	// Step 2: Debounce filter (for rising edge)
	// TON: Q=TRUE only if rawInverted stays TRUE for DebounceTime continuously
	// rawInverted=FALSE immediately sets Q=FALSE (falling edge is unfiltered)
	// Note: To also filter the falling edge, add TOF -- not implemented currently
	#tonDebounce(IN := #rawInverted,
	             PT := #DebounceTime);

	IF #DebounceTime > T#0ms THEN
	    #State := #tonDebounce.Q;   // Filtered signal
	ELSE
	    #State := #rawInverted;     // Unfiltered (when DebounceTime=0)
	END_IF;

	// Step 3: Edge detection (compare with previous scan)
	#RisingEdge := #State AND NOT #prevState;
	#FallingEdge := NOT #State AND #prevState;
	#prevState := #State;

END_FUNCTION_BLOCK

FUNCTION_BLOCK "FB_SpindleControl"
{ S7_Optimized_Access := 'TRUE' }
VERSION : 3.0
// =============================================================================
// 07_SpindleControl.scl
// FB_SpindleControl -- Spindle speed control (simplified)
//
// Purpose:
//   Controls the spindle in velocity mode using MC_MoveVelocity (PTO output).
//   VFD run direction: CW only -- no direction pin.
//   RunForward signal enables VFD run.
//
// â”€â”€â”€â”€â”€â”€â”€â”€â”€â”€â”€â”€â”€â”€â”€â”€â”€â”€â”€â”€â”€â”€â”€â”€â”€â”€â”€â”€â”€â”€â”€â”€â”€â”€â”€â”€â”€â”€â”€â”€â”€â”€â”€â”€â”€â”€â”€â”€â”€â”€â”€â”€â”€â”€â”€â”€â”€â”€â”€â”€â”€â”€â”€â”€â”€â”€â”€â”€â”€â”€â”€â”€â”€â”€â”€â”€â”€
// OPERATING RULES (enforced by the CALLER, not by this FB):
//
//   1. Set SetSpeed while RunCmd = FALSE.
//   2. Set RunCmd = TRUE  â†’ MC_MoveVelocity starts + RunForward goes TRUE.
//      Keep RunCmd TRUE for the entire run.
//   3. To stop:  set RunCmd = FALSE  â†’ RunForward goes FALSE, PTO halts.
//      Do NOT touch SetSpeed during stop.
//   4. To change speed:
//        a. RunCmd = FALSE  (spindle coasts / stops on VFD ramp)
//        b. Write new SetSpeed
//        c. RunCmd = TRUE   (spindle restarts at new speed)
//
// This FB does NOT add any delays or intermediate states.
// Timing handshakes (coast-down waits, PTO stabilise, etc.) are the CALLER's
// responsibility if they are needed.
//
// â”€â”€â”€â”€â”€â”€â”€â”€â”€â”€â”€â”€â”€â”€â”€â”€â”€â”€â”€â”€â”€â”€â”€â”€â”€â”€â”€â”€â”€â”€â”€â”€â”€â”€â”€â”€â”€â”€â”€â”€â”€â”€â”€â”€â”€â”€â”€â”€â”€â”€â”€â”€â”€â”€â”€â”€â”€â”€â”€â”€â”€â”€â”€â”€â”€â”€â”€â”€â”€â”€â”€â”€â”€â”€â”€â”€â”€
// Speed calculation:
//   effectiveSpeed = CLAMP(SetSpeed, MinSpeed, MaxSpeed)
//   PTO conversion: velocity (pulse/s) = effectiveRPM Ã— 500 / 60
//   MinSpeed and MaxSpeed are read from DB_Spindle.
//
// Error codes:
//   16#0502 -- MC_MoveVelocity runtime error
//
// States (Diag_SpindleState):
//   0   = IDLE     -- RunCmd FALSE, all outputs safe
//   20  = RUNNING  -- RunCmd TRUE, PTO active, RunForward TRUE
//   999 = ERROR    -- cleared by AckError or Reset
//
// Change log:
//   2026-05-09  Complete rewrite: RunCmd level input replaces Start/Stop edges.
//               Removed STARTING and STOPPING delay states and mid-run
//               velocity-change handshake.  Caller owns all sequencing.
//   2026-05-09  Previous version: 4-state machine (was 7-state before that).
// =============================================================================
   VAR_INPUT
      Enable : Bool;   // Drive power enable -- from bDrivesEnable; stays TRUE during normal operation
      RunCmd : Bool;   // Level signal: TRUE = run, FALSE = stop/idle.   Set speed first, then raise RunCmd.   Lower RunCmd to stop; do not change speed while RunCmd is TRUE.
      SetSpeed : Real;   // Commanded speed in RPM (set while RunCmd = FALSE)
      SpeedOverride : Real;   // Speed override % (100 = normal speed)
      Reset : Bool;   // Full system reset -- clears ERROR, returns to IDLE
      AckError : Bool;   // Acknowledge spindle error only (no full system reset needed)
   END_VAR

   VAR_OUTPUT
      Running : Bool;   // TRUE while RunCmd is TRUE and no error
      AtSpeed : Bool;   // TRUE when actual speed is within SpeedTolerance of commanded
      ActualSpeed : Real;   // Measured speed (RPM)
      CommandedSpeed : Real;   // Override-applied target speed (RPM)
      Error : Bool;   // Error active
      ErrorID : Word;   // Error code
      RunForward : Bool;   // VFD Run Forward digital output -- mirrors RunCmd (except in ERROR)
   END_VAR

   VAR_IN_OUT
      Axis_Spindle {InstructionName := 'TO_PositioningAxis'; LibVersion := '8.0'} : TO_PositioningAxis;   // Spindle Technology Object
   END_VAR

   VAR
      state : Int;   // 0 = IDLE, 20 = RUNNING, 999 = ERROR Speed calculation
      effectiveRPM : Real;   // RPM after override and clamping
      targetVelocity : Real;   // Velocity in pulse/s sent to MC_MoveVelocity Motion FB instances
      MC_Power_Inst {InstructionName := 'MC_Power'; LibVersion := '8.0'} : MC_Power;
      MC_MoveVelocity_Inst {InstructionName := 'MC_MoveVelocity'; LibVersion := '8.0'} : MC_MoveVelocity;   // Internal execute flag
      bMoveVelExec : Bool;   // AtSpeed helpers
      speedDiff : Real;
      speedPercent : Real;   // AckError edge detection
      prevAck : Bool;
      ackEdge : Bool;
   END_VAR


BEGIN

	// =========================================================================
	// 1. EDGE DETECTION
	// =========================================================================
	#ackEdge := #AckError AND NOT #prevAck;
	#prevAck := #AckError;

	// =========================================================================
	// 2. RESET (full system reset -- takes priority over everything)
	// =========================================================================
	IF #Reset THEN
	    #state := 0;
	    #Error := FALSE;
	    #ErrorID := 0;
	    #bMoveVelExec := FALSE;
	    #RunForward := FALSE;
	END_IF;

	// =========================================================================
	// 3. SPEED CALCULATION (runs every scan)
	// =========================================================================
	#effectiveRPM := #SetSpeed * (#SpeedOverride / 100.0);
	IF #effectiveRPM < "DB_Spindle".MinSpeed THEN
	    #effectiveRPM := "DB_Spindle".MinSpeed;
	END_IF;
	IF #effectiveRPM > "DB_Spindle".MaxSpeed THEN
	    #effectiveRPM := "DB_Spindle".MaxSpeed;
	END_IF;
	#CommandedSpeed := #effectiveRPM;
	#targetVelocity := #effectiveRPM * 500.0 / 60.0;  // RPM â†’ pulse/s

	// =========================================================================
	// 4. STATE MACHINE
	// =========================================================================
	CASE #state OF

	        // -----------------------------------------------------------------
	        // STATE 0: IDLE
	        // All outputs safe.  Transition to RUNNING when RunCmd goes TRUE.
	        // -----------------------------------------------------------------
	    0:
	        #Running := FALSE;
	        #AtSpeed := FALSE;
	        #bMoveVelExec := FALSE;
	        #RunForward := FALSE;

	        IF #RunCmd THEN
	            #bMoveVelExec := TRUE;  // pre-load velocity; RunForward still FALSE
	            #state := 10;
	        END_IF;

	        // -----------------------------------------------------------------
	        // STATE 10: PRELOAD
	        // Execute TRUE so the PTO frequency is stable before the VFD is
	        // enabled.  RunForward stays FALSE this scan; transitions to RUNNING
	        // on the very next scan.
	        // -----------------------------------------------------------------
	    10:
	        #Running := FALSE;
	        #AtSpeed := FALSE;
	        #bMoveVelExec := TRUE;
	        #RunForward := FALSE;
	        #state := 20;

	        // -----------------------------------------------------------------
	        // STATE 20: RUNNING
	        // RunCmd TRUE â†’ MC_MoveVelocity active, RunForward TRUE.
	        // The CALLER is responsible for sequencing (speed-change stops,
	        // coast-down waits, PTO-stabilise delays, etc.).
	        // Transition back to IDLE when RunCmd goes FALSE.
	        // -----------------------------------------------------------------
	    20:
	        IF NOT #RunCmd THEN
	            // Caller dropped RunCmd â†’ stop immediately
	            #Running := FALSE;
	            #AtSpeed := FALSE;
	            #bMoveVelExec := FALSE;
	            #RunForward := FALSE;
	            #state := 0;

	        ELSE
	            // Normal running
	            #Running := TRUE;
	            #bMoveVelExec := TRUE;
	            #RunForward := TRUE;

	            // AtSpeed check
	            #speedDiff := ABS(#ActualSpeed - #effectiveRPM);
	            #speedPercent := 0.0;
	            IF #effectiveRPM > 1.0 THEN
	                #speedPercent := (#speedDiff / #effectiveRPM) * 100.0;
	            END_IF;
	            #AtSpeed := (#speedPercent <= "DB_Spindle".SpeedTolerance);

	            // MC_MoveVelocity error check
	            IF #MC_MoveVelocity_Inst.Error THEN
	                #ErrorID := 16#0502;
	                #bMoveVelExec := FALSE;
	                #RunForward := FALSE;
	                "DB_Diagnostic".Spindle_TO_ErrorID := #MC_MoveVelocity_Inst.ErrorID;
	                "DB_Diagnostic".TO_ErrorText := "FC_TO_ErrorText"(Code := #MC_MoveVelocity_Inst.ErrorID);
	                "DB_Diagnostic".Error_Text := CONCAT(IN1 := 'Spindle move failed: ',
	                                                     IN2 := "DB_Diagnostic".TO_ErrorText);
	                "DB_Diagnostic".Error_Code := #ErrorID;
	                // Single-writer: report via queue -> FB_AlarmManager latches DB_Error and
	                // drives DB_HMI.ErrorText through the mirror. (The old direct ErrorText
	                // write here was overwritten by the mirror one scan later and the error
	                // never reached DB_Error/history at all.)
	                "FC_ReportError"(Code := #ErrorID,
	                                 Details := "DB_Diagnostic".Error_Text,
	                                 Source := 'Spindle');
	                "DB_HMI".ErrorDetail := CONCAT(IN1 := 'TO:', IN2 := "DB_Diagnostic".TO_ErrorText);
	                "DB_HMI".ErrorDetail_ES := CONCAT(IN1 := 'TO:', IN2 := "DB_Diagnostic".TO_ErrorText);
	                #state := 999;
	            END_IF;
	        END_IF;

	        // -----------------------------------------------------------------
	        // STATE 999: ERROR
	        // AckError: clears spindle error, returns to IDLE.
	        // Reset:    handled above (takes priority, clears everything).
	        // -----------------------------------------------------------------
	    999:
	        #Error := TRUE;
	        #Running := FALSE;
	        #AtSpeed := FALSE;
	        #bMoveVelExec := FALSE;
	        #RunForward := FALSE;

	        IF #ackEdge THEN
	            #Error := FALSE;
	            #ErrorID := 0;
	            #state := 0;
	            // DB_HMI error text is owned by FB_AlarmManager (mirror) â€” Ack clears it
	            // there; STATE_STOPPED clears ErrorDetail. No HMI writes from this FB.
	        END_IF;

	END_CASE;

	// =========================================================================
	// 5. MC_ FUNCTION BLOCK CALLS (every scan)
	// =========================================================================
	#MC_Power_Inst(
	               Axis := #Axis_Spindle,
	               Enable := #Enable
	);
	#MC_MoveVelocity_Inst(
	                      Axis := #Axis_Spindle,
	                      Execute := #bMoveVelExec,
	                      Velocity := #targetVelocity,
	                      Direction := 1              // CW only -- no direction pin
	);

	// Actual speed: TO velocity (pulse/s) â†’ RPM
	#ActualSpeed := ABS(#Axis_Spindle.ActualVelocity) * 60.0 / 500.0;

	// =========================================================================
	// 6. WRITE STATUS TO DB_Spindle (read by HMI and other FBs)
	// =========================================================================
	"DB_Spindle".IsRunning := #Running;
	"DB_Spindle".AtSpeed := #AtSpeed;
	"DB_Spindle".ActualSpeed := #ActualSpeed;
	"DB_Spindle".CommandedSpeed := #CommandedSpeed;
	"DB_Spindle".Error := #Error;
	"DB_Spindle".ErrorID := #ErrorID;

	// Diagnostics (written every scan for watch-table tracing)
	"DB_Spindle".Diag_SpindleState := #state;    // 0=Idle, 10=Preload, 20=Running, 999=Error
	"DB_Spindle".Diag_MoveVelBusy := #MC_MoveVelocity_Inst.Busy;
	"DB_Spindle".Diag_MoveVelInVel := #MC_MoveVelocity_Inst.InVelocity;


END_FUNCTION_BLOCK

DATA_BLOCK "TO_AxisX"
{InstructionName := 'TO_PositioningAxis';
 LibVersion := '8.0';
 S7_Optimized_Access := 'TRUE' }
AUTHOR : SIMATIC
FAMILY : BasicMC
NAME : TO_PosAx
VERSION : 8.0
NON_RETAIN
TO_PositioningAxis

BEGIN
   Header.VersionMaj := 8;
   Header.VersionMin := 0;
   Actor.InverseDirection := FALSE;
   Actor.Interface.PTO := 16#88E1_0109;
   Actor.DriveParameter.PulsesPerDriveRevolution := 2048;
   Sensor[1].ActiveHoming.DigitalInputAddress.RID := 16#0200_0001;
   Sensor[1].ActiveHoming.DigitalInputAddress.AREA := 16#81;
   Sensor[1].ActiveHoming.DigitalInputAddress.OFFSET := 4;
   Sensor[1].ActiveHoming.HomePositionOffset := 10.0;
   Mechanics.LeadScrew := 1.0;
   DynamicLimits.MaxVelocity := 40.0;
   DynamicLimits.MinVelocity := 0.001;
   DynamicDefaults.Acceleration := 153.8423;
   DynamicDefaults.Deceleration := 184.6108;
   DynamicDefaults.EmergencyDeceleration := 3999.9;
   DynamicDefaults.Jerk := 512.8076;
   PositionLimits_SW.Active := FALSE;
   PositionLimits_SW.MinPosition := -50.0;
   PositionLimits_SW.MaxPosition := 350.0;
   PositionLimits_HW.Active := TRUE;
   PositionLimits_HW.MinSwitchAddress.RID := 16#0200_0001;
   PositionLimits_HW.MinSwitchAddress.AREA := 16#81;
   PositionLimits_HW.MinSwitchAddress.OFFSET := 9;
   PositionLimits_HW.MaxSwitchAddress.RID := 16#0200_0001;
   PositionLimits_HW.MaxSwitchAddress.AREA := 16#81;
   PositionLimits_HW.MaxSwitchAddress.OFFSET := 10;
   Homing.AutoReversal := TRUE;
   Homing.ApproachDirection := FALSE;
   Homing.ApproachVelocity := 30.0;
   Homing.ReferencingVelocity := 10.0;

END_DATA_BLOCK

FUNCTION "FC_CylinderDispatch" : Void
{ S7_Optimized_Access := 'TRUE' }
VERSION : 0.1
// =============================================================================
// FC_CylinderDispatch -- Routes manual cylinder commands to the selected cylinder
// =============================================================================
//
// Reads command fields from DB_Manual.SelectedCylinder and related fields,
// writes them to the corresponding DB_CylinderX instance, then mirrors
// status back to DB_Manual.SelCyl_* for HMI display.
//
// Called from OB1 AFTER all cylinder FB calls so status reflects the current scan.
// Commands have a one-scan delay relative to the HMI write -- imperceptible in practice.
//
// ADDING A CYLINDER:
//   1. Add DATA_BLOCK "DB_CylinderN" in 02_DataBlocks.scl
//   2. Add sensor FB calls + DB_CylinderN() call + solenoid outputs in OB1
//   3. Copy CASE 1 block below, change all DB_Cylinder1 â†’ DB_CylinderN,
//      and update SelCyl_Name string.
// =============================================================================

BEGIN

	// Apply cylinder config on rising edge of Btn_ApplyType (PositioningMode + Tolerance)
	IF "DB_Manual".Btn_ApplyType AND NOT "DB_Manual".prevBtn_ApplyType THEN
	    CASE "DB_Manual".SelectedCylinder OF
	        1:
	            "DB_Cylinder_BackSupport".PositioningMode := INT_TO_BYTE("DB_Manual".SelCyl_SetType);
	            "DB_Cylinder_BackSupport".Tolerance := "DB_Manual".Cyl_Tolerance;
	        2:
	            "DB_Cylinder_SheetHolder".PositioningMode := INT_TO_BYTE("DB_Manual".SelCyl_SetType);
	            "DB_Cylinder_SheetHolder".Tolerance := "DB_Manual".Cyl_Tolerance;
	        3:
	            "DB_Cylinder_ToolHeadLock".PositioningMode := INT_TO_BYTE("DB_Manual".SelCyl_SetType);
	            "DB_Cylinder_ToolHeadLock".Tolerance := "DB_Manual".Cyl_Tolerance;
	        4:
	            "DB_Cylinder_MandrelLock".PositioningMode := INT_TO_BYTE("DB_Manual".SelCyl_SetType);
	            "DB_Cylinder_MandrelLock".Tolerance := "DB_Manual".Cyl_Tolerance;
	    END_CASE;
	END_IF;
	"DB_Manual".prevBtn_ApplyType := "DB_Manual".Btn_ApplyType;

	CASE "DB_Manual".SelectedCylinder OF

	    1: // BackSupport -- linear ruler, PositioningMode=3
	        "DB_Manual".SelCyl_Name := 'BackSupport';
	        "DB_Cylinder_BackSupport".Cmd_ExtendFull := "DB_Manual".Btn_CylExtendFull;
	        "DB_Cylinder_BackSupport".Cmd_RetractFull := "DB_Manual".Btn_CylRetractFull;
	        "DB_Cylinder_BackSupport".Cmd_GotoPos := "DB_Manual".Btn_CylGotoPos;
	        "DB_Cylinder_BackSupport".TargetPos := "DB_Manual".Cyl_TargetPos;
	        "DB_Manual".SelCyl_State := "DB_Cylinder_BackSupport".State;
	        "DB_Manual".SelCyl_StateText := "DB_Cylinder_BackSupport".StateText;
	        "DB_Manual".SelCyl_AtSetpoint := "DB_Cylinder_BackSupport".AtSetpoint;
	        "DB_Manual".SelCyl_AtRetract := "DB_Cylinder_BackSupport".AtRetract;
	        "DB_Manual".SelCyl_AtTarget := FALSE;
	        "DB_Manual".SelCyl_PosError := 0.0;
	        "DB_Manual".SelCyl_Error := "DB_Cylinder_BackSupport".Error;
	        "DB_Manual".SelCyl_ErrorID := "DB_Cylinder_BackSupport".ErrorID;
	        "DB_Manual".SelCyl_ActualPos := "DB_Cylinder_LinearRuler_BackSupport".Value;
	        "DB_Manual".SelCyl_Type := BYTE_TO_INT("DB_Cylinder_BackSupport".PositioningMode);
	        "DB_Manual".SelCyl_Toleranse := "DB_Cylinder_BackSupport".Tolerance;
	        "DB_Manual".SelCyl_MaxPos := "DB_Cylinder_BackSupport".MaxPos;
	        "DB_Manual".SelCyl_MinPos := "DB_Cylinder_BackSupport".MinPos;

	    2: // SheetHolder -- no sensor, PositioningMode=0
	        "DB_Manual".SelCyl_Name := 'SheetHolder';
	        "DB_Cylinder_SheetHolder".Cmd_ExtendFull := "DB_Manual".Btn_CylExtendFull;
	        "DB_Cylinder_SheetHolder".Cmd_RetractFull := "DB_Manual".Btn_CylRetractFull;
	        "DB_Cylinder_SheetHolder".Cmd_GotoPos := "DB_Manual".Btn_CylGotoPos;
	        "DB_Cylinder_SheetHolder".TargetPos := "DB_Manual".Cyl_TargetPos;
	        "DB_Manual".SelCyl_State := "DB_Cylinder_SheetHolder".State;
	        "DB_Manual".SelCyl_StateText := "DB_Cylinder_SheetHolder".StateText;
	        "DB_Manual".SelCyl_AtSetpoint := "DB_Cylinder_SheetHolder".AtSetpoint;
	        "DB_Manual".SelCyl_AtRetract := "DB_Cylinder_SheetHolder".AtRetract;
	        "DB_Manual".SelCyl_AtTarget := FALSE;
	        "DB_Manual".SelCyl_PosError := 0.0;
	        "DB_Manual".SelCyl_Error := "DB_Cylinder_SheetHolder".Error;
	        "DB_Manual".SelCyl_ErrorID := "DB_Cylinder_SheetHolder".ErrorID;
	        "DB_Manual".SelCyl_ActualPos := 0.0;
	        "DB_Manual".SelCyl_Type := BYTE_TO_INT("DB_Cylinder_SheetHolder".PositioningMode);
	        "DB_Manual".SelCyl_Toleranse := "DB_Cylinder_SheetHolder".Tolerance;
	        "DB_Manual".SelCyl_MaxPos := "DB_Cylinder_SheetHolder".MaxPos;
	        "DB_Manual".SelCyl_MinPos := "DB_Cylinder_SheetHolder".MinPos;

	    3: // ToolHeadLock -- magnetic sensor, PositioningMode=1
	        // CRITICAL: This cylinder locks the tool head. When extended (Sol_A=TRUE),
	        // tool axis movement is blocked at the process level.
	        // Manual extend/retract is allowed here for commissioning only.
	        "DB_Manual".SelCyl_Name := 'ToolHeadLock';
	        "DB_Cylinder_ToolHeadLock".Cmd_ExtendFull := "DB_Manual".Btn_CylExtendFull;
	        "DB_Cylinder_ToolHeadLock".Cmd_RetractFull := "DB_Manual".Btn_CylRetractFull;
	        "DB_Cylinder_ToolHeadLock".Cmd_GotoPos := "DB_Manual".Btn_CylGotoPos;
	        "DB_Cylinder_ToolHeadLock".TargetPos := "DB_Manual".Cyl_TargetPos;
	        "DB_Manual".SelCyl_State := "DB_Cylinder_ToolHeadLock".State;
	        "DB_Manual".SelCyl_StateText := "DB_Cylinder_ToolHeadLock".StateText;
	        "DB_Manual".SelCyl_AtSetpoint := "DB_Cylinder_ToolHeadLock".AtSetpoint;
	        "DB_Manual".SelCyl_AtRetract := "DB_Cylinder_ToolHeadLock".AtRetract;
	        "DB_Manual".SelCyl_AtTarget := FALSE;
	        "DB_Manual".SelCyl_PosError := 0.0;
	        "DB_Manual".SelCyl_Error := "DB_Cylinder_ToolHeadLock".Error;
	        "DB_Manual".SelCyl_ErrorID := "DB_Cylinder_ToolHeadLock".ErrorID;
	        "DB_Manual".SelCyl_ActualPos := 0.0;
	        "DB_Manual".SelCyl_Type := BYTE_TO_INT("DB_Cylinder_ToolHeadLock".PositioningMode);
	        "DB_Manual".SelCyl_Toleranse := "DB_Cylinder_ToolHeadLock".Tolerance;
	        "DB_Manual".SelCyl_MaxPos := "DB_Cylinder_ToolHeadLock".MaxPos;
	        "DB_Manual".SelCyl_MinPos := "DB_Cylinder_ToolHeadLock".MinPos;

	    4: // MandrelLock -- no sensor, PositioningMode=0
	        "DB_Manual".SelCyl_Name := 'MandrelLock';
	        "DB_Cylinder_MandrelLock".Cmd_ExtendFull := "DB_Manual".Btn_CylExtendFull;
	        "DB_Cylinder_MandrelLock".Cmd_RetractFull := "DB_Manual".Btn_CylRetractFull;
	        "DB_Cylinder_MandrelLock".Cmd_GotoPos := "DB_Manual".Btn_CylGotoPos;
	        "DB_Cylinder_MandrelLock".TargetPos := "DB_Manual".Cyl_TargetPos;
	        "DB_Manual".SelCyl_State := "DB_Cylinder_MandrelLock".State;
	        "DB_Manual".SelCyl_StateText := "DB_Cylinder_MandrelLock".StateText;
	        "DB_Manual".SelCyl_AtSetpoint := "DB_Cylinder_MandrelLock".AtSetpoint;
	        "DB_Manual".SelCyl_AtRetract := "DB_Cylinder_MandrelLock".AtRetract;
	        "DB_Manual".SelCyl_AtTarget := FALSE;
	        "DB_Manual".SelCyl_PosError := 0.0;
	        "DB_Manual".SelCyl_Error := "DB_Cylinder_MandrelLock".Error;
	        "DB_Manual".SelCyl_ErrorID := "DB_Cylinder_MandrelLock".ErrorID;
	        "DB_Manual".SelCyl_ActualPos := 0.0;
	        "DB_Manual".SelCyl_Type := BYTE_TO_INT("DB_Cylinder_MandrelLock".PositioningMode);
	        "DB_Manual".SelCyl_Toleranse := "DB_Cylinder_MandrelLock".Tolerance;
	        "DB_Manual".SelCyl_MaxPos := "DB_Cylinder_MandrelLock".MaxPos;
	        "DB_Manual".SelCyl_MinPos := "DB_Cylinder_MandrelLock".MinPos;

	    ELSE:
	        // Unknown selector -- show N/A, no commands routed
	        "DB_Manual".SelCyl_Name := '---';
	        "DB_Manual".SelCyl_State := 0;
	        "DB_Manual".SelCyl_StateText := 'N/A';
	        "DB_Manual".SelCyl_AtSetpoint := FALSE;
	        "DB_Manual".SelCyl_AtRetract := FALSE;
	        "DB_Manual".SelCyl_AtTarget := FALSE;
	        "DB_Manual".SelCyl_PosError := 0.0;
	        "DB_Manual".SelCyl_Error := FALSE;
	        "DB_Manual".SelCyl_ErrorID := 16#0000;
	        "DB_Manual".SelCyl_ActualPos := 0.0;
	        "DB_Manual".SelCyl_Type := 0;
	        "DB_Manual".SelCyl_Toleranse := 0.0;
	        "DB_Manual".SelCyl_MaxPos := 0.0;
	        "DB_Manual".SelCyl_MinPos := 0.0;

	END_CASE;

END_FUNCTION

ORGANIZATION_BLOCK "Startup"
TITLE = "PLC Startup - Load Configuration"
{ S7_Optimized_Access := 'TRUE' }
VERSION : 1.0
// -----------------------------------------------------------------------------
// OB100 -- Startup Organization Block
// Runs ONCE on PLC power-up, transition to RUN mode, or program download.
// Calls FC_LoadConfig -- do not add anything else here; keep everything inside FC.
// -----------------------------------------------------------------------------
   VAR_TEMP
      tempRetVal : Int;
   END_VAR


BEGIN

	"FC_LoadConfig"();

END_ORGANIZATION_BLOCK

DATA_BLOCK "fbProcess"
{ S7_Optimized_Access := 'TRUE' }
VERSION : 0.1
NON_RETAIN
// Instance Data Block for FB_Process
"FB_Process"

BEGIN

END_DATA_BLOCK

DATA_BLOCK "DB_fbSpindle"
{ S7_Optimized_Access := 'TRUE' }
VERSION : 0.1
NON_RETAIN
// -----------------------------------------------------------------------------
// DB_fbSpindle -- FB_SpindleControl instance (NO LONGER CALLED IN OB1)
// Spindle is now controlled exclusively via fbSpindleControl inside FB_Process (fbProcess DB).
// This DB is retained so TIA Portal does not lose the symbol. Do not call from OB1.
// DB_Spindle (separate) â†’ spindle status + HMI outputs (IsRunning, AtSpeed, etc.)
// -----------------------------------------------------------------------------
"FB_SpindleControl"

BEGIN

END_DATA_BLOCK

DATA_BLOCK "DB_Cylinder_BackSupport"
{ S7_Optimized_Access := 'TRUE' }
VERSION : 0.5
NON_RETAIN
// =============================================================================
// PNEUMATIC CYLINDER INSTANCE DATA BLOCKS
// =============================================================================
// Instances of FBs defined in 09_Sensors_Actuators.scl.
// HMI reads/writes these DBs directly -- no separate interface DB needed.
//
// Cylinder map:
//   CylDiag[1] = DB_BackSupport    (full stroke, PositioningMode=0; ruler HW removed on this machine)
//   CylDiag[2] = DB_SheetHolder    (no sensor, PositioningMode=0, ValveType=1)
//   CylDiag[3] = DB_ToolHeadLock   (magnetic sensor, PositioningMode=1, safety lock)
//   CylDiag[4] = DB_MandrelLock    (no sensor, PositioningMode=0)
// =============================================================================
// =============================================================================
// BACKSUPPORT CYLINDER (CylDiag[1]) -- Full stroke, PositioningMode=0
//
// Ruler hardware removed on this machine. CMD=40 triggers a full extension;
// AtSetpoint fires after Timeout_Extend. 5/3 blocked-center valve holds mechanically.
// DB_Cylinder_LinearRuler_BackSupport and OB1 ruler call are retained for future use
// if the ruler is re-fitted (switch PositioningMode back to 3 and re-enable in OB1).
// TIA tags:  Output_Cyl_Backsupport_SolA/B
// =============================================================================
// -----------------------------------------------------------------------------
// DB_BackSupport -- FB_CylinderControl instance
// PositioningMode=0 (full stroke, timed), ValveType=2 (5/3 blocked center)
//
// HMI WRITABLE:   Cmd_ExtendFull, Cmd_RetractFull
// HMI READ-ONLY:  Sol_A, Sol_B, State, StateText, AtSetpoint, Error, ErrorID
// CONNECTED IN OB1: SafetyOK, RulerValue, RulerValid (ruler inputs ignored in Mode=0)
// To re-enable ruler: change PositioningMode to 3 and restore ruler tuning fields below.
// -----------------------------------------------------------------------------
"FB_CylinderControl"

BEGIN
   ValveType := 2;
   Timeout_Extend := T#1S_500MS;
   Timeout_Retract := T#10S;
   PositioningMode := 0;

END_DATA_BLOCK

DATA_BLOCK "DB_Cylinder_Sen_BackSupport_Setpt"
{ S7_Optimized_Access := 'TRUE' }
VERSION : 0.1
NON_RETAIN
"FB_DigitalSensor"

BEGIN
   DebounceTime := T#10MS;

END_DATA_BLOCK

DATA_BLOCK "DB_Cylinder_LinearRuler_BackSupport"
{ S7_Optimized_Access := 'TRUE' }
VERSION : 0.1
NON_RETAIN
// -----------------------------------------------------------------------------
// DB_Cylinder_LinearRuler_BackSupport -- FB_AnalogSensor instance
// Analog linear ruler for BackSupport cylinder position feedback.
// Connected in OB1: AI_LinearRuler_BackSupport â†’ RulerValue/RulerValid on cylinder FB.
// Calibration is set in FC_LoadConfig Section 6; HMI can adjust at runtime.
// InvertSignal=TRUE: 0V = full extend (~300mm), ~10V = retracted (0mm).
// -----------------------------------------------------------------------------
"FB_AnalogSensor"

BEGIN
   Raw_Max := 31433;
   Phys_Max := 300.0;
   InvertSignal := TRUE;
   Hi_Limit := 295.0;
   Lo_Limit := 5.0;

END_DATA_BLOCK

DATA_BLOCK "DB_Cylinder_SheetHolder"
{ S7_Optimized_Access := 'TRUE' }
VERSION : 0.1
NON_RETAIN
// =============================================================================
// SHEETHOLDER CYLINDER (CylDiag[2]) -- No sensor, full stroke (PositioningMode=0)
//
// TIA Portal tags: Output_Cyl_SheetHolder_SolA  (Sol_B not wired -- ValveType=1)
// =============================================================================
// -----------------------------------------------------------------------------
// DB_SheetHolder -- FB_CylinderControl instance
// ValveType=1 (5/2 spring return, single solenoid):
//   Sol_A=TRUE  â†’ piston extends (sheet held).
//   Sol_A=FALSE â†’ spring retracts. Power loss = safe retract.
// PositioningMode=0: no sensor -- full stroke, timeout = done, no error.
// -----------------------------------------------------------------------------
"FB_CylinderControl"

BEGIN
   ValveType := 1;
   Timeout_Extend := T#5S;
   Timeout_Retract := T#5S;
   PositioningMode := 0;

END_DATA_BLOCK

DATA_BLOCK "DB_Cylinder_ToolHeadLock"
{ S7_Optimized_Access := 'TRUE' }
VERSION : 0.3
NON_RETAIN
// =============================================================================
// TOOLHEADLOCK CYLINDER (CylDiag[3]) -- Magnetic sensor (PositioningMode=1, safety lock)
//
// LOCK BEHAVIOR (implemented in FB_Process):
//   EXTEND (Sol_A ON)  : states STATE_RUNNING (20) and STATE_PAUSED (25) only.
//   RETRACT (spring)   : all other states -- power loss also retracts (spring return).
//
// SEQUENCE GATES (FB_Process checks sensor before state transition):
//   Before entering RUNNING     : STATE_LOCK_EXTEND_WAIT (17) -- AtSetpoint OR 2s timer fallback.
//   Before TOOL_CHANGE / homing : STATE_LOCK_RETRACT_WAIT (29) -- 2s timer (no retract sensor).
//
// TIA Portal tags: In_Cyl_ToolHeadLock_AtSetpoint, Output_Cyl_ToolHeadLock_SolA
//                  (Sol_B not wired -- ValveType=1)
// =============================================================================
// -----------------------------------------------------------------------------
// DB_ToolHeadLock -- FB_CylinderControl instance
// ValveType=1 (5/2 spring return, single solenoid):
//   Sol_A=TRUE  â†’ piston extends (locked).
//   Sol_A=FALSE â†’ spring retracts (unlocked). Power loss = safe retract.
// Sen_AtSetpoint confirms lock fully engaged; Timeout_Extend=T#6S is error fallback.
// State 17 in FB_Process transitions when AtSetpoint=TRUE (sensor only; no fallback timer in FB_Process).
// Timeout_Extend in this DB is the only timer -- if sensor does not confirm within 6s, CylFB reports Error.
// -----------------------------------------------------------------------------
"FB_CylinderControl"

BEGIN
   ValveType := 1;
   Timeout_Extend := T#6S;
   Timeout_Retract := T#2S;
   PositioningMode := 1;

END_DATA_BLOCK

DATA_BLOCK "DB_Cylinder_Sen_ToolHeadLock_Setpt"
{ S7_Optimized_Access := 'TRUE' }
VERSION : 0.1
NON_RETAIN
"FB_DigitalSensor"

BEGIN
   DebounceTime := T#10MS;

END_DATA_BLOCK

DATA_BLOCK "DB_Cylinder_MandrelLock"
{ S7_Optimized_Access := 'TRUE' }
VERSION : 0.1
NON_RETAIN
// =============================================================================
// MANDRELLOCK CYLINDER (CylDiag[4]) -- No sensor, full stroke (PositioningMode=0)
//
// TIA Portal tags: Output_Cyl_MandrelLock_SolA, Output_Cyl_MandrelLock_SolB
// =============================================================================
// -----------------------------------------------------------------------------
// DB_MandrelLock -- FB_CylinderControl instance
// -----------------------------------------------------------------------------
"FB_CylinderControl"

BEGIN
   ValveType := 1;
   Timeout_Extend := T#5S;
   Timeout_Retract := T#5S;
   PositioningMode := 0;

END_DATA_BLOCK

FUNCTION "FC_ContactorControl" : Void
{ S7_Optimized_Access := 'TRUE' }
VERSION : 0.1
// -----------------------------------------------------------------------------
// FC_ContactorControl -- Manages physical drive contactor and enable outputs.
//
// Safety condition: no output is active without E-Stop OK (physical or bypass).
// On error (MachineError): contactors and enable signals are dropped.
// Enable interlock: Enable can only be active when the associated contactor is also on.
//
// Sequence: Contactor ON â†’ Enable ON â†’ MC_Power.Enable := TRUE â†’ drive ready
// -----------------------------------------------------------------------------
   VAR_TEMP
      eStopOK : Bool;   // E-Stop cleared (physical or bypass)
      drivePermit : Bool;   // Only E-Stop controls contactor permission
      modePermit : Bool;   // State-based interlock: prevents contactor in STATE_STOPPED (0) only
   END_VAR


BEGIN

	#eStopOK := "Safety_Estop" OR "DB_HMI".Bypass_EStop;
	#drivePermit := #eStopOK;  // Only E-Stop cuts contactor power -- NC/PNP/errors do NOT cut power

	// Mode interlock: contactors blocked only in STATE_STOPPED (0).
	// STATE_ERROR (999) is ALLOWED so contactors stay on after a PNP/NC halt --
	// operator can jog away from limit zone without a full restart cycle.
	// In auto states (>=10), FB_Process writes Btn_Contactor_* programmatically.
	#modePermit := "DB_HMI".MachineState > 0;

	// Contactor outputs
	"Output_Contactor_X" := "DB_HMI".Btn_Contactor_X AND #drivePermit AND #modePermit;
	"Output_Contactor_Z" := "DB_HMI".Btn_Contactor_Z AND #drivePermit AND #modePermit;
	"Output_Contactor_Tool" := "DB_HMI".Btn_Contactor_Tool AND #drivePermit AND #modePermit;
	"Output_Contactor_Spindle" := "DB_HMI".Btn_Contactor_Spindle AND #drivePermit AND #modePermit;

	// Enable outputs -- associated contactor must also be on (interlock)
	"Output_Enable_X" := "DB_HMI".Btn_Enable_X AND "DB_HMI".Btn_Contactor_X AND #drivePermit AND #modePermit;
	"Output_Enable_Z" := "DB_HMI".Btn_Enable_Z AND "DB_HMI".Btn_Contactor_Z AND #drivePermit AND #modePermit;

	// HMI lamp feedback
	"DB_HMI".Contactor_X_On := "Output_Contactor_X";
	"DB_HMI".Contactor_Z_On := "Output_Contactor_Z";
	"DB_HMI".Contactor_Tool_On := "Output_Contactor_Tool";
	"DB_HMI".Contactor_Spindle_On := "Output_Contactor_Spindle";
	"DB_HMI".Enable_X_On := "Output_Enable_X";
	"DB_HMI".Enable_Z_On := "Output_Enable_Z";

END_FUNCTION

ORGANIZATION_BLOCK "Main"
TITLE = "Main Program Sweep (Cycle)"
{ S7_Optimized_Access := 'TRUE' }
VERSION : 0.1
// -----------------------------------------------------------------------------
// OB1 -- Main cyclic loop entry point
// -----------------------------------------------------------------------------
   VAR_TEMP
      tempRetVal : Int;
   END_VAR


BEGIN

	// =========================================================================
	// E-STOP DUAL CHANNEL -- Must run BEFORE all other FB calls
	// =========================================================================
	// Safety_Estop_Ch1 and Safety_Estop_Ch2: physical DI (%I) addresses in TIA Portal tag table.
	// Safety_Estop: Marker (%M) -- computed combined signal.
	"DB_fbEStop"(Ch1_NC := "Safety_Estop_Ch1",
	             Ch2_NO := "Safety_Estop_Ch2",
	             DiscrepancyTimeout := "DB_MachineConfig".Timeout_EStopDiscrep);

	// Combined E-Stop signal: safe when both channels are closed
	"Safety_Estop" := "DB_fbEStop".EStop_OK;

	// HMI status update
	"DB_HMI".EStop_Ch1_OK := "Safety_Estop_Ch1";
	"DB_HMI".EStop_Ch2_OK := "Safety_Estop_Ch2";
	"DB_HMI".EStop_Discrepancy := "DB_fbEStop".Discrepancy;

	// Discrepancy alarm: triggered once after timeout â†’ FB_AlarmManager generates 16#0406
	IF "DB_fbEStop".DiscrepancyAlarm THEN
	    "FC_ReportError"(Code := 16#0406,
	                     Details := 'E-Stop contact discrepancy - check wiring/contacts',
	                     Source := 'Safety');
	END_IF;

	// Main process state machine
	"fbProcess"(
	            Panel_Start    := "Panel_Start_A" AND "Panel_Start_B",
	            Panel_Stop     := "Panel_Stop",
	            Panel_Pause    := "Panel_Pause",
	            Panel_Reset    := "Panel_Reset",
	            Rem_Start      := FALSE,
	            Rem_Stop       := FALSE,
	            EStop_OK       := "Safety_Estop",
	            Door_Closed    := "Safety_Door",
	            AirPressure_OK := "Safety_Air",
	            HW_NC_X_Min    := "Limit_NC_X_Min",
	            HW_NC_X_Max    := "Limit_NC_X_Max",
	            HW_NC_Z_Min    := "Limit_NC_Z_Min",
	            HW_NC_Z_Max    := "Limit_NC_Z_Max",
	            HW_PNP_X_Min   := "Limit_PNP_X_Min",
	            HW_PNP_X_Max   := "Limit_PNP_X_Max",
	            HW_PNP_Z_Min   := "Limit_PNP_Z_Min",
	            HW_PNP_Z_Max   := "Limit_PNP_Z_Max",
	            Axis_X         := "TO_AxisX",
	            Axis_Z         := "TO_AxisZ",
	            Axis_Tool      := "TO_AxisTool",
	            Axis_Spindle   := "TO_AxisSpindle"
	);

	// =========================================================================
	// PNEUMATIC CYLINDERS
	// Sensor FBs must run BEFORE their cylinder FB (State must be updated first).
	// FC_CylinderDispatch must run AFTER all cylinder FBs (mirrors status to DB_Manual).
	//
	// Cylinder map:
	//   CylDiag[1] = DB_BackSupport  (full stroke, PositioningMode=0; ruler HW removed) -- SelectedCylinder=1
	//   CylDiag[2] = DB_SheetHolder  (no sensor, PositioningMode=0, ValveType=1) -- SelectedCylinder=2
	//   CylDiag[3] = DB_ToolHeadLock (magnetic sensor, PositioningMode=1) -- SelectedCylinder=3
	//   CylDiag[4] = DB_MandrelLock  (no sensor, PositioningMode=0) -- SelectedCylinder=4
	// =========================================================================

	// â”€â”€ BackSupport (CylDiag[1]) -- full stroke, PositioningMode=0 â”€â”€â”€â”€â”€â”€â”€â”€â”€â”€â”€
	// Ruler HW removed on this machine. Ruler FB call and RulerValue/RulerValid inputs
	// are retained so Mode=3 can be restored later by changing PositioningMode in
	// DB_Cylinder_BackSupport. In Mode=0 the cylinder FB ignores these inputs.
	"DB_Cylinder_LinearRuler_BackSupport"(AI_Raw := "AI_LinearRuler_Backsupport");
	"DB_Cylinder_Sen_BackSupport_Setpt"(RawInput := "In_Cyl_BackSupport_AtSetpoint");
	"DB_Cylinder_BackSupport"(
	                          SafetyOK       := "Safety_Estop" OR "DB_HMI".Bypass_EStop,
	                          Sen_AtSetpoint := "DB_Cylinder_Sen_BackSupport_Setpt".State,
	                          RulerValue     := "DB_Cylinder_LinearRuler_BackSupport".Value,
	                          RulerValid     := "DB_Cylinder_LinearRuler_BackSupport".Valid
	);
	"Output_Cyl_Backsupport_SolA" := "DB_Cylinder_BackSupport".Sol_A;
	// Sol_B: normal FB output OR CMD=41 Param=1 override (holds retract solenoid independently)
	"Output_Cyl_Backsupport_SolB" := "DB_Cylinder_BackSupport".Sol_B
	OR "DB_Cylinder_BackSupport".SolB_Cmd41;
	// Atmosphere valve: energised by CMD=41 Param=1, de-energised by Param=2 or process stop
	"Output_Cyl_Backsupport_SolAtmosphere" := "DB_Cylinder_BackSupport".SolAtmo_Cmd;
	"DB_Diagnostic".CylDiag[1].State := "DB_Cylinder_BackSupport".State;
	"DB_Diagnostic".CylDiag[1].Pos := "DB_Cylinder_LinearRuler_BackSupport".Value;
	"DB_Diagnostic".CylDiag[1].Sol_A := "DB_Cylinder_BackSupport".Sol_A;
	"DB_Diagnostic".CylDiag[1].Sol_B := "DB_Cylinder_BackSupport".Sol_B;
	"DB_Diagnostic".CylDiag[1].Error := "DB_Cylinder_BackSupport".Error;
	"DB_Diagnostic".CylDiag[1].ErrorID := "DB_Cylinder_BackSupport".ErrorID;

	// â”€â”€ SheetHolder (CylDiag[2]) -- no sensor, PositioningMode=0, ValveType=1 â”€â”€
	"DB_Cylinder_SheetHolder"(
	                          SafetyOK := "Safety_Estop" OR "DB_HMI".Bypass_EStop
	);
	"Output_Cyl_SheetHolder_SolA" := "DB_Cylinder_SheetHolder".Sol_A;
	"DB_Diagnostic".CylDiag[2].State := "DB_Cylinder_SheetHolder".State;
	"DB_Diagnostic".CylDiag[2].Pos := 0.0;
	"DB_Diagnostic".CylDiag[2].Sol_A := "DB_Cylinder_SheetHolder".Sol_A;
	"DB_Diagnostic".CylDiag[2].Sol_B := "DB_Cylinder_SheetHolder".Sol_B;
	"DB_Diagnostic".CylDiag[2].Error := "DB_Cylinder_SheetHolder".Error;
	"DB_Diagnostic".CylDiag[2].ErrorID := "DB_Cylinder_SheetHolder".ErrorID;

	// â”€â”€ ToolHeadLock (CylDiag[3]) -- magnetic sensor, PositioningMode=1, ValveType=1 â”€
	// Cmd_Extend is written every scan by FB_Process based on machine state:
	//   EXTEND  : STATE_RUNNING (20), STATE_PAUSED (25), STATE_LOCK_EXTEND_WAIT (17)
	//   RETRACT : all other states (spring return; includes ERROR, STOPPED, homing, tool change)
	// State 17 transitions when AtSetpoint confirms lock engaged, or after 2s timer fallback.
	"DB_Cylinder_Sen_ToolHeadLock_Setpt"(RawInput := "In_Cyl_ToolHeadLock_AtSetpoint");
	"DB_Cylinder_ToolHeadLock"(
	                           SafetyOK       := "Safety_Estop" OR "DB_HMI".Bypass_EStop,
	                           Sen_AtSetpoint := "DB_Cylinder_Sen_ToolHeadLock_Setpt".State
	);
	"Output_Cyl_ToolHeadLock_SolA" := "DB_Cylinder_ToolHeadLock".Sol_A;
	"DB_Diagnostic".CylDiag[3].State := "DB_Cylinder_ToolHeadLock".State;
	"DB_Diagnostic".CylDiag[3].Pos := 0.0;
	"DB_Diagnostic".CylDiag[3].Sol_A := "DB_Cylinder_ToolHeadLock".Sol_A;
	"DB_Diagnostic".CylDiag[3].Sol_B := "DB_Cylinder_ToolHeadLock".Sol_B;
	"DB_Diagnostic".CylDiag[3].Error := "DB_Cylinder_ToolHeadLock".Error;
	"DB_Diagnostic".CylDiag[3].ErrorID := "DB_Cylinder_ToolHeadLock".ErrorID;

	// â”€â”€ MandrelLock (CylDiag[4]) -- no sensor, PositioningMode=0 â”€â”€â”€â”€â”€â”€â”€â”€â”€â”€â”€â”€â”€
	// Cmd_Extend driven by FB_Process in STATE_SHEET_WAIT phase 2 (clamp during sheet loading).
	// SafetyOK override: keep MandrelLock extended (workpiece clamped) during RUNNING (20),
	// PAUSED (25), STOPPING (18), and ERROR (999) even if E-Stop fires. The workpiece must not
	// be released while the spindle is still coasting after an E-Stop -- ejecting the sheet at
	// speed is more hazardous than holding it clamped. Retract is triggered explicitly by
	// bMandrelRetractPulse when the operator acknowledges or resets from STATE_ERROR (lines
	// 2244/2256/2271/1477 in 06_MainProcess.scl), and Cmd_Extend is cleared every scan in
	// STATE_STOPPED (line 1514). All error-exit paths fire the retract pulse before reaching
	// STOPPED, so the mandrel cannot remain permanently extended.
	"DB_Cylinder_MandrelLock"(
	                          SafetyOK := "Safety_Estop" OR "DB_HMI".Bypass_EStop OR
	                          ("DB_HMI".MachineState = 20) OR  // STATE_RUNNING
	                          ("DB_HMI".MachineState = 25) OR  // STATE_PAUSED
	                          ("DB_HMI".MachineState = 18) OR  // STATE_STOPPING
	                          ("DB_HMI".MachineState = 999)    // STATE_ERROR: hold clamp until explicit Ack/Reset
	);
	"Output_Cyl_MandrelLock_SolA" := "DB_Cylinder_MandrelLock".Sol_A;
	"DB_Diagnostic".CylDiag[4].State := "DB_Cylinder_MandrelLock".State;
	"DB_Diagnostic".CylDiag[4].Pos := 0.0;
	"DB_Diagnostic".CylDiag[4].Sol_A := "DB_Cylinder_MandrelLock".Sol_A;
	"DB_Diagnostic".CylDiag[4].Error := "DB_Cylinder_MandrelLock".Error;
	"DB_Diagnostic".CylDiag[4].ErrorID := "DB_Cylinder_MandrelLock".ErrorID;

	// Cylinder manual command dispatch (selected cylinder â†’ DB_Manual SelCyl_* status)
	// Must run AFTER all cylinder FB calls so status reflects the current scan.
	"FC_CylinderDispatch"();

	// Contactor and enable outputs: FC_ContactorControl is called at the END of
	// FB_Process (in sync with the state machine) -- NOT here. ITEM-37: the
	// duplicate OB1 call was removed; nothing between fbProcess and this point
	// writes any input the FC depends on (Btn_Contactor_*, Bypass_EStop,
	// MachineState, Safety_Estop), so one call per scan is sufficient.

	// Automatically update tool slot angles based on slot count
	"FC_ToolAngleCalc"();

END_ORGANIZATION_BLOCK

